(*
:Description: Wire-format body schema for FB_Metrics push frames.

Encoded as a single byte at offset +0x03 of ST_PushMetricAggHeader. The
body of the frame is always sample_count * sample_size bytes; this enum
tells the receiver how to interpret each fixed-size slot.

Mapped from the locked IEC type at the first Observe() call. Numerics
(SINT..LREAL incl. unsigned) collapse to ``eNumeric`` and are widened
to LREAL (sample_size = 8). BOOL / discrete / strings keep their raw
sample size.
*)
TYPE INTERNAL E_MetricBodySchema :
(
    eUnknown            := 0,
    eBool               := 1,    // body: sample_count * 1 byte
    eNumeric            := 2,    // body: sample_count * 8 bytes (LREAL, widened)
    eDiscrete           := 3,    // body: sample_count * sample_size raw bytes (BYTE/WORD/DWORD/LWORD/ENUM)
    eString             := 4,    // body: sample_count * sample_size UTF-8 bytes (zero-padded fixed)
    eWstring            := 5,    // body: sample_count * sample_size UTF-16LE bytes (zero-padded fixed)
    eNumericAggregated  := 6     // body: sample_count * popcount(stat_mask) LREALs in bit-order
                                 // — see E_MetricStat for the bit assignments
) BYTE;
END_TYPE

(* stored: Version 1.1.0.1, ProductVersion 3.1.4026.18
   DUT E_MetricBodySchema: Id {96d11b28-f297-0796-3243-7238571e2874} *)
